TYPE udtLogging :
STRUCT
	StartLog	:	BOOL;
	LogID		:	INT;
END_STRUCT
END_TYPE

(* stored: Version 1.1.0.1, ProductVersion 3.1.4024.11
   DUT udtLogging: Id {1d5b9ad3-62a5-4bd1-958c-aaa607d6f8e8} *)
